PROGRAM MAIN
VAR
	USVCyclicComm : PS_Q4_DcUpsEC_Cyclic_3;
	USVParamComm  : PS_Q4_DcUpsEC_Param_1;
	
	arrInputPD	AT%I* : ARRAY [0..30] OF WORD;	// Connect Multilink of TxPDO here
	
END_VAR

USVCyclicComm(xActivate:=TRUE,arrInputPD:=arrInputPD);
// USVParamComm();

END_PROGRAM

(* stored: Version 1.1.0.1, ProductVersion 3.1.4026.18
   POU MAIN: Id {85bd1b41-5549-4d90-a836-6937aec40ea7}, SpecialFunc None *)
